RoboDK station: Curved_Conv.rdk

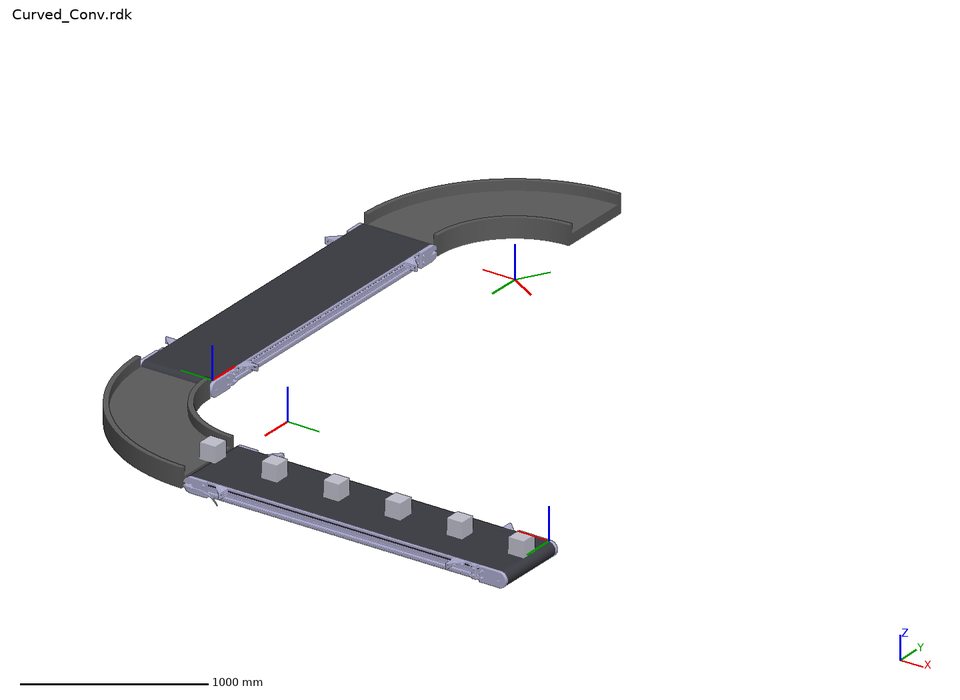
[picture v0: the station drawn from its stored meshes, robots at their saved joint values, targets as dots, program paths as lines]
Station Curved_Conv (saved by RoboDK 5.6.0). Poses are relative to the parent item; angles as X-Y-Z fixed-axis rotations.
  - frame Convetor 1 at (2020, 440, 0) mm, rotated rx 0 ry 0 rz 180 deg
    - robot Conv_Mech1: 1 axes
        modified DH rows (alpha deg, a mm, theta deg, d mm): 0, 0, 0, 0 linear
        base shift (0, 0, 0) mm, rotated rx 0 ry 90 rz 0 deg
        joint limits [-500000] to [500000]; home [0]; saved at [0]
      - frame Frame_Conv1 at (0, 0, 0) mm
        - object box 1 at (40, 200, 50) mm, rotated rx 0 ry 0 rz -180 deg, size 100 x 100 x 100 mm, geometry from box.sld
        - object box 2 at (440, 200, 50) mm, rotated rx 0 ry 0 rz -180 deg, size 100 x 100 x 100 mm, geometry from box.sld
        - object box 3 at (840, 200, 50) mm, rotated rx 0 ry 0 rz -180 deg, size 100 x 100 x 100 mm, geometry from box.sld
        - object box 4 at (1240, 200, 50) mm, rotated rx 0 ry 0 rz -180 deg, size 100 x 100 x 100 mm, geometry from box.sld
        - object box 5 at (1640, 200, 50) mm, rotated rx 0 ry 0 rz -180 deg, size 100 x 100 x 100 mm, geometry from box.sld
        - object box 6 at (2040, 200, 50) mm, rotated rx 0 ry 0 rz -180 deg, size 100 x 100 x 100 mm, geometry from box.sld
  - frame Conveyor 2 at (-560, 1010, 0) mm, rotated rx 0 ry 0 rz 90 deg
    - robot Conv_Mech2: 1 axes
        modified DH rows (alpha deg, a mm, theta deg, d mm): 0, 0, 0, 0 linear
        base shift (0, 0, 0) mm, rotated rx 0 ry 90 rz 0 deg
        joint limits [-500000] to [500000]; home [0]; saved at [0]
      - frame Frame_Conv2 at (0, 0, 0) mm
  - frame Curved_Conv at (-40, 960, -80) mm, rotated rx 0 ry 0 rz -90 deg
    - robot Curved_Conv_Mech: 1 axes
        modified DH rows (alpha deg, a mm, theta deg, d mm): 0, 0, 0, 0
        joint limits [-200000] to [0]; home [0]; saved at [0]
      - frame Frame_CurveConv at (0, 0, 0) mm
  - program Reset (2 instructions, listed below)
  - folder Python
    - Python program Run_Conveyor_Curve (listed below)
    - Python program Run_Conveyor1 (listed below)
    - Python program Run_Conveyor2 (listed below)
    - Python program Reset_All_Mechanism (listed below)
    - Python program Switch_Obj_ref (listed below)
    - Python program Run_Conveyor_Curve2 (listed below)
  - program Main (5 instructions, listed below)
  - frame Curved_Conv2 at (-40, 3065, -80) mm, rotated rx 0 ry 0 rz -180 deg
    - robot Curved_Conv_Mech2: 1 axes
        modified DH rows (alpha deg, a mm, theta deg, d mm): 0, 0, 0, 0
        joint limits [-200000] to [0]; home [0]; saved at [-4890]
      - frame Frame_CurveConv2 at (0, 0, 0) mm

--- program Reset (robot Conv_Mech1) ---
  Call Reset_All_Mechanism
  Replace objects

--- Python program Run_Conveyor_Curve ---
# Type help("robolink") or help("robodk") for more information
# Press F5 to run the script
# Documentation: https://robodk.com/doc/en/RoboDK-API.html
# Reference:     https://robodk.com/doc/en/PythonAPI/index.html
# Note: It is not required to keep a copy of this file, your python script is saved with the station
from robolink import *    # RoboDK API
from robodk import *      # Robot toolbox
RDK = Robolink()

#Set the travel of the conveyors for each iterations
PART_ROTATION_ANGLE = -30

#Declaration of the conveyor object
Conv_curved = RDK.Item('Curved_Conv_Mech',itemtype=ITEM_TYPE_ROBOT)

#setSpeed(speed_linear, speed_joints, accel_linear, accel_joints),
#Must adjust to match the linear conveyors speed
Conv_curved.setSpeed(7,7,7,7)

#If the conveyor exist, move it to the declared value.
if Conv_curved.Valid():
    Conv_curved.MoveJ(Conv_curved.Joints() + PART_ROTATION_ANGLE)

--- Python program Run_Conveyor1 ---
# Type help("robolink") or help("robodk") for more information
# Press F5 to run the script
# Documentation: https://robodk.com/doc/en/RoboDK-API.html
# Reference:     https://robodk.com/doc/en/PythonAPI/index.html
# Note: It is not required to keep a copy of this file, your python script is saved with the station
from robolink import *    # RoboDK API
from robodk import *      # Robot toolbox
RDK = Robolink()

#Set the travel of the conveyors for each iterations
PART_TRAVEL_MM = 400

#Declaration of the conveyor object
Conv_mechanism1 = RDK.Item('Conv_Mech1',itemtype=ITEM_TYPE_ROBOT)

#If the conveyor exist, move it to the declared value.
if Conv_mechanism1.Valid():
    Conv_mechanism1.MoveJ(Conv_mechanism1.Joints() + PART_TRAVEL_MM)

--- Python program Run_Conveyor2 ---
# Type help("robolink") or help("robodk") for more information
# Press F5 to run the script
# Documentation: https://robodk.com/doc/en/RoboDK-API.html
# Reference:     https://robodk.com/doc/en/PythonAPI/index.html
# Note: It is not required to keep a copy of this file, your python script is saved with the station
from robolink import *    # RoboDK API
from robodk import *      # Robot toolbox
RDK = Robolink()

#Set the travel of the conveyors for each iterations
PART_TRAVEL_MM = 400

#Declaration of the conveyor object
Conv_mechanism2 = RDK.Item('Conv_Mech2',itemtype=ITEM_TYPE_ROBOT)

#If the conveyor exist, move it to the declared value.
if Conv_mechanism2.Valid():
    Conv_mechanism2.MoveJ(Conv_mechanism2.Joints() + PART_TRAVEL_MM)

--- Python program Reset_All_Mechanism ---
# Type help("robolink") or help("robodk") for more information
# Press F5 to run the script
# Documentation: https://robodk.com/doc/en/RoboDK-API.html
# Reference:     https://robodk.com/doc/en/PythonAPI/index.html
# Note: It is not required to keep a copy of this file, your python script is saved with the station
from robolink import *    # RoboDK API
from robodk import *      # Robot toolbox
RDK = Robolink()

#This program reinitialize every mechanisms in the list to position 0
MECHANISM_LIST = ["Conv_Mech1","Conv_Mech2","Curved_Conv_Mech"]

for i in range(len(MECHANISM_LIST)):
    MECHANISM_NAME=MECHANISM_LIST[i]
    mechanism = RDK.Item(MECHANISM_NAME,itemtype=ITEM_TYPE_ROBOT)
    if mechanism.Valid():
        mechanism.setJoints([0])

--- Python program Switch_Obj_ref ---
# Type help("robolink") or help("robodk") for more information
# Press F5 to run the script
# Documentation: https://robodk.com/doc/en/RoboDK-API.html
# Reference:     https://robodk.com/doc/en/PythonAPI/index.html
# Note: It is not required to keep a copy of this file, your python script is saved with the station
from robolink import *    # RoboDK API
from robodk import *      # Robot toolbox
RDK = Robolink()

#Declaration of the frames
frame_conv1 = RDK.Item('Frame_Conv1',itemtype=ITEM_TYPE_FRAME)
frame_conv2 = RDK.Item('Frame_Conv2',itemtype=ITEM_TYPE_FRAME)
frame_curve = RDK.Item('Frame_CurveConv',itemtype=ITEM_TYPE_FRAME)
frame_curve2 = RDK.Item('Frame_CurveConv2',itemtype=ITEM_TYPE_FRAME)

#Declaration of the child frames
obj_list1 = frame_conv1.Childs()
obj_list2 = frame_curve.Childs()
obj_list3 = frame_conv2.Childs()  # Add this line to get objects in Curve2

for item in obj_list1:
    print("\nframe_conv1 positions")
    print(item.PoseAbs()) #If you want to see the Abs pos matrix of the object
    if item.PoseAbs()[0,3] < 0: #[0,3] refer to line 0 column 3 in the pos matrix, so the X position
        item.setParentStatic(frame_curve)

for item in obj_list2:
    print("\nframe_curve 1 positions")
    print(item.PoseAbs()) #If you want to see the Abs pos matrix of the object
    if item.PoseAbs()[1,3] > 900: #[1,3] refer to line 1 column 3 in the pos matrix, so the Y position
        item.setParentStatic(frame_conv2)

for item in obj_list3:
    #print("\nframe_curve 2 positions")
    print(item.PoseAbs())
    if item.PoseAbs()[1,3] > 2920:  # Check proximity to Curve2
        item.setParentStatic(frame_curve2)

--- Python program Run_Conveyor_Curve2 ---
# Type help("robolink") or help("robodk") for more information
# Press F5 to run the script
# Documentation: https://robodk.com/doc/en/RoboDK-API.html
# Reference:     https://robodk.com/doc/en/PythonAPI/index.html
# Note: It is not required to keep a copy of this file, your python script is saved with the station
from robolink import *    # RoboDK API
from robodk import *      # Robot toolbox
RDK = Robolink()

#Set the travel of the conveyors for each iterations
PART_ROTATION_ANGLE = -30

#Declaration of the conveyor object
Conv_curved2 = RDK.Item('Curved_Conv_Mech2',itemtype=ITEM_TYPE_ROBOT)

#setSpeed(speed_linear, speed_joints, accel_linear, accel_joints),
#Must adjust to match the linear conveyors speed
Conv_curved2.setSpeed(7,7,7,7)

#If the conveyor exist, move it to the declared value.
if Conv_curved2.Valid():
    Conv_curved2.MoveJ(Conv_curved2.Joints() + PART_ROTATION_ANGLE)

--- program Main (robot Conv_Mech1) ---
  Call Switch_Obj_ref
  Run Run_Conveyor1
  Run Run_Conveyor_Curve
  Call Run_Conveyor2
  Run Run_Conveyor_Curve2
